(* PLC project FbdPinsProject *)

PROGRAM FbdPins

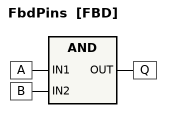
(* FBD diagram, written out as Structured Text *)
Q := A AND B;
END_PROGRAM

CONFIGURATION Config
  RESOURCE Res ON PLC
  END_RESOURCE
END_CONFIGURATION
